// TwinCAT 3 PLC project Untitled1
// ProgramVersion: 3.1.4024.0
// libraries:
//   Tc2_Standard, * (Beckhoff Automation GmbH)
//   Tc2_System, * (Beckhoff Automation GmbH)
//   Tc3_Module, * (Beckhoff Automation GmbH)
//   TcUnit,1.2.0.0,www.tcunit.org
// project tree:
//   / PlcTask.TcTTO
//   POUs/ MAIN.TcPOU, FB_Sum.TcPOU
//   Tests/ FB_Sum_Test.TcPOU, PRG_TEST.TcPOU
// real-time tasks:
//   TASK PlcTask: cycle T#10ms, priority 20, ADS port 350

CONFIGURATION Untitled1
    RESOURCE PLC ON TwinCAT3
        TASK PlcTask(INTERVAL := T#10ms, PRIORITY := 20);
        PROGRAM MAIN WITH PlcTask : MAIN;
        PROGRAM PRG_TEST WITH PlcTask : PRG_TEST;
    END_RESOURCE
END_CONFIGURATION

// ---- POUs/MAIN.TcPOU
PROGRAM MAIN
VAR
END_VAR

END_PROGRAM

// ---- Tests/PRG_TEST.TcPOU
PROGRAM PRG_TEST
VAR
    fbSum_Test : FB_Sum_Test; // This is our test suite
END_VAR

TcUnit.RUN();

END_PROGRAM

// ---- Tests/FB_Sum_Test.TcPOU
FUNCTION_BLOCK FB_Sum_Test EXTENDS TcUnit.FB_TestSuite
VAR_INPUT
END_VAR
VAR_OUTPUT
END_VAR
VAR
END_VAR

TwoPlusTwoEqualsFour();
ZeroPlusZeroEqualsZero();

METHOD TwoPlusTwoEqualsFour
VAR
    Sum : FB_Sum;
    Result : UINT;
    ExpectedSum : UINT := 4;
	
	ExpectedProp : BOOL;
END_VAR
TEST('TwoPlusTwoEqualsFour');
 
Sum(one := 2, two := 2, result => Result);
 
AssertEquals(Expected := ExpectedSum,
             Actual := Result,
             Message := 'The calculation is not correct');
			 
//This line of code makes my pc crash, I mean crash HARD! As in Blue-Screen-Of-Death crash...
AssertEquals(Expected := ExpectedProp,
             Actual := Sum.Prop,
             Message := 'Testing prop');			 
 
TEST_FINISHED();
END_METHOD

METHOD ZeroPlusZeroEqualsZero
VAR
    Sum : FB_Sum;
    Result : UINT;
    ExpectedSum : UINT := 0;
END_VAR
TEST('ZeroPlusZeroEqualsZero');
 
Sum(one := 0, two := 0, result => Result);
 
AssertEquals(Expected := ExpectedSum,
             Actual := Result,
             Message := 'The calculation is not correct');
 
TEST_FINISHED();
END_METHOD

END_FUNCTION_BLOCK

// ---- POUs/FB_Sum.TcPOU
FUNCTION_BLOCK FB_Sum
VAR_INPUT
	one : UINT;
    two : UINT;
END_VAR
VAR_OUTPUT
    result : UINT;
END_VAR
VAR
	_prop:BOOL:=FALSE;
END_VAR

PROPERTY Prop : BOOL
GET
Prop := _prop;
END_GET
SET
_prop:=Prop;
END_SET
END_PROPERTY

END_FUNCTION_BLOCK
